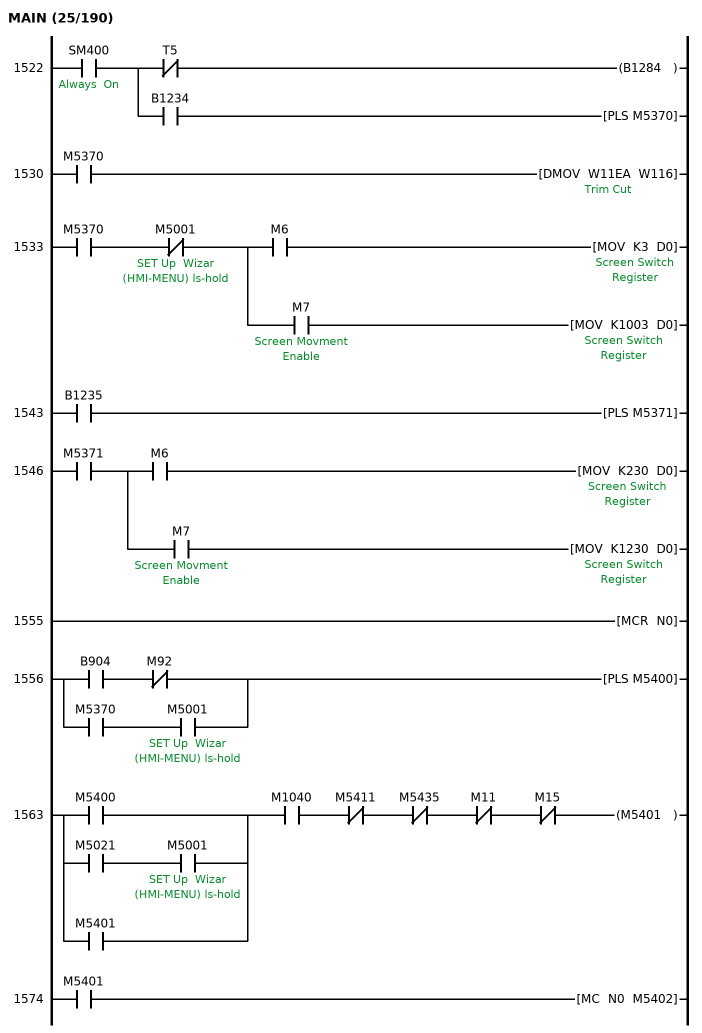
[picture p24: ladder of MAIN, rungs at steps 1522 to 1574]
1522  LD      SM400  ; Always  On
      MPS
      ANI     T5
      OUT     B1284
      MPP
      AND     B1234
      PLS     M5370
1530  LD      M5370
      DMOV    W11EA W116
1533  LD      M5370
      ANI     M5001  ; SET Up  Wizar (HMI-MENU) ls-hold
      MPS
      AND     M6
      MOV     K3 D0
      MPP
      AND     M7  ; Screen Movment Enable
      MOV     K1003 D0
1543  LD      B1235
      PLS     M5371
1546  LD      M5371
      MPS
      AND     M6
      MOV     K230 D0
      MPP
      AND     M7  ; Screen Movment Enable
      MOV     K1230 D0
1555  MCR     N0
1556  LD      B904
      ANI     M92
      LD      M5370
      AND     M5001  ; SET Up  Wizar (HMI-MENU) ls-hold
      ORB
      PLS     M5400
1563  LD      M5400
      LD      M5021
      AND     M5001  ; SET Up  Wizar (HMI-MENU) ls-hold
      ORB
      OR      M5401
      AND     M1040
      ANI     M5411
      ANI     M5435
      ANI     M11
      ANI     M15
      OUT     M5401
1574  LD      M5401
      MC      N0 M5402
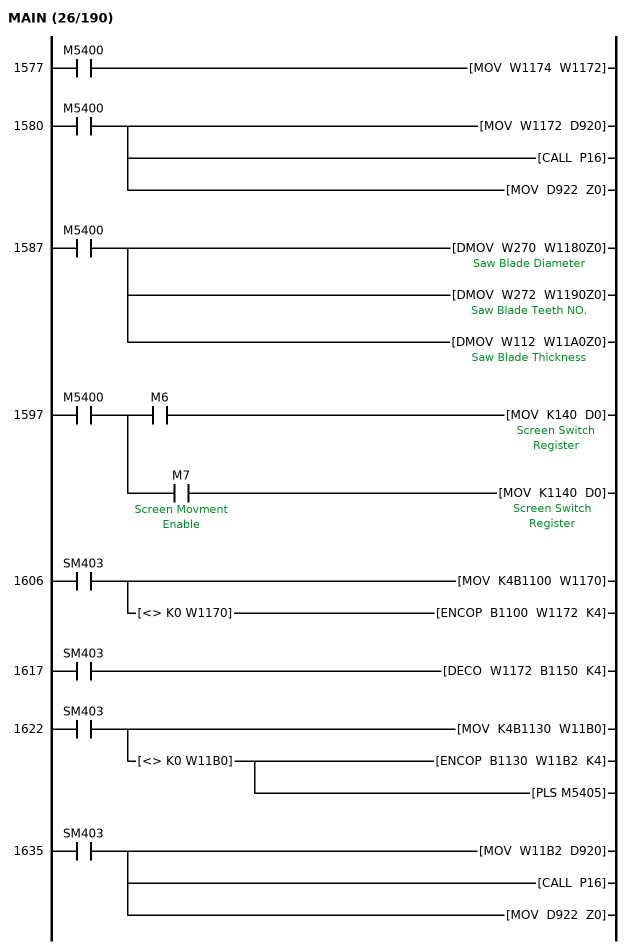
1577  LD      M5400
      MOV     W1174 W1172
1580  LD      M5400
      MOV     W1172 D920
      CALL    P16
      MOV     D922 Z0
1587  LD      M5400
      DMOV    W270 W1180Z0  ; Saw Blade Diameter
      DMOV    W272 W1190Z0  ; Saw Blade Teeth NO.
      DMOV    W112 W11A0Z0  ; Saw Blade Thickness
1597  LD      M5400
      MPS
      AND     M6
      MOV     K140 D0
      MPP
      AND     M7  ; Screen Movment Enable
      MOV     K1140 D0
1606  LD      SM403
      MOV     K4B1100 W1170
      AND<>   K0 W1170
      ENCOP   B1100 W1172 K4
1617  LD      SM403
      DECO    W1172 B1150 K4
1622  LD      SM403
      MOV     K4B1130 W11B0
      AND<>   K0 W11B0
      ENCOP   B1130 W11B2 K4
      PLS     M5405
1635  LD      SM403
      MOV     W11B2 D920
      CALL    P16
      MOV     D922 Z0
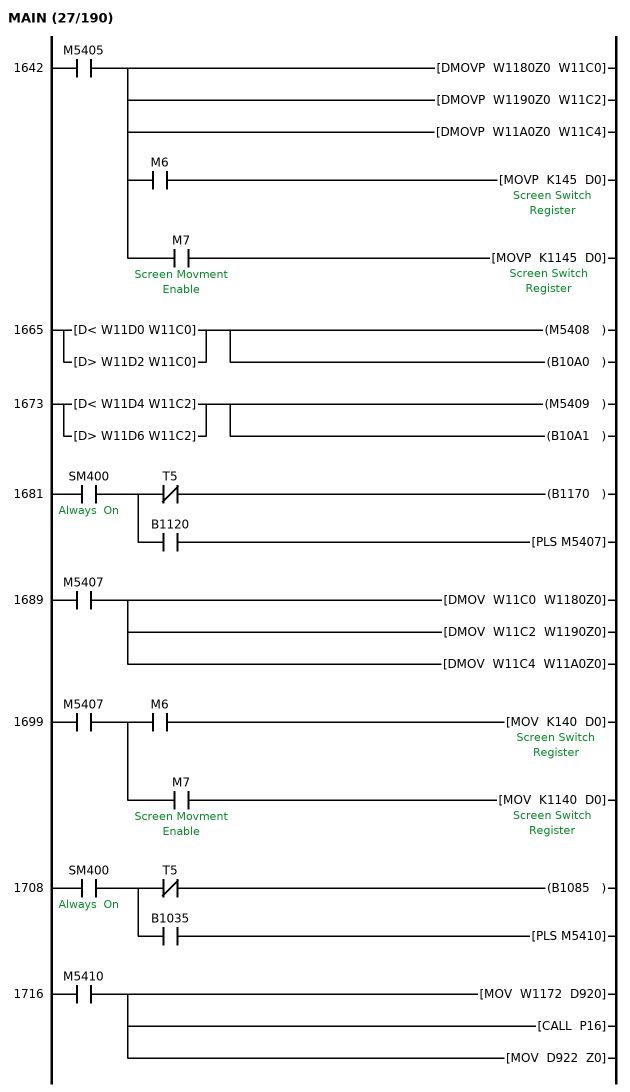
1642  LD      M5405
      DMOVP   W1180Z0 W11C0
      DMOVP   W1190Z0 W11C2
      DMOVP   W11A0Z0 W11C4
      MPS
      AND     M6
      MOVP    K145 D0
      MPP
      AND     M7  ; Screen Movment Enable
      MOVP    K1145 D0
1665  LDD<    W11D0 W11C0
      ORD>    W11D2 W11C0
      OUT     M5408
      OUT     B10A0
1673  LDD<    W11D4 W11C2
      ORD>    W11D6 W11C2
      OUT     M5409
      OUT     B10A1
1681  LD      SM400  ; Always  On
      MPS
      ANI     T5
      OUT     B1170
      MPP
      AND     B1120
      PLS     M5407
1689  LD      M5407
      DMOV    W11C0 W1180Z0
      DMOV    W11C2 W1190Z0
      DMOV    W11C4 W11A0Z0
1699  LD      M5407
      MPS
      AND     M6
      MOV     K140 D0
      MPP
      AND     M7  ; Screen Movment Enable
      MOV     K1140 D0
1708  LD      SM400  ; Always  On
      MPS
      ANI     T5
      OUT     B1085
      MPP
      AND     B1035
      PLS     M5410
1716  LD      M5410
      MOV     W1172 D920
      CALL    P16
      MOV     D922 Z0
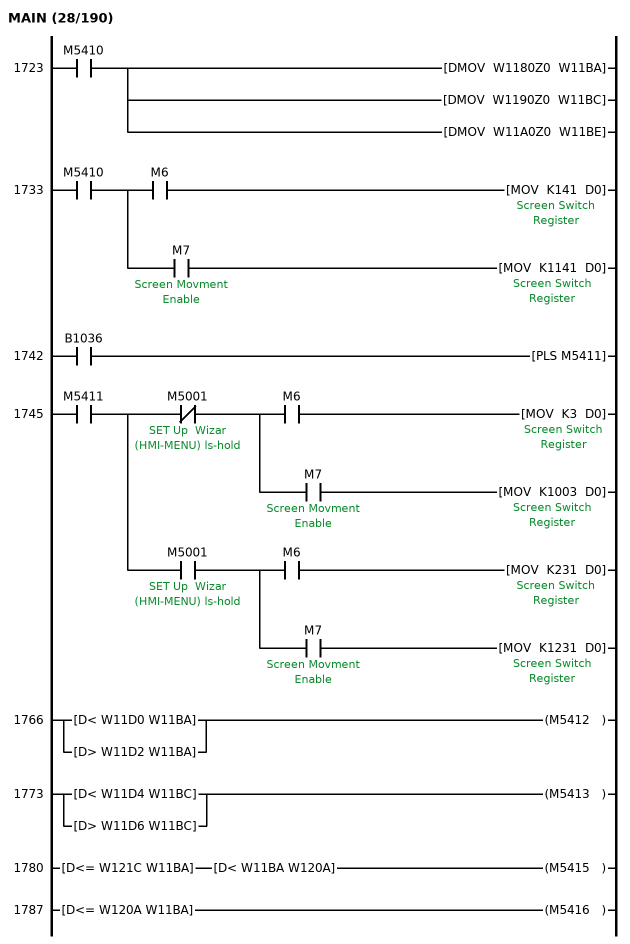
1723  LD      M5410
      DMOV    W1180Z0 W11BA
      DMOV    W1190Z0 W11BC
      DMOV    W11A0Z0 W11BE
1733  LD      M5410
      MPS
      AND     M6
      MOV     K141 D0
      MPP
      AND     M7  ; Screen Movment Enable
      MOV     K1141 D0
1742  LD      B1036
      PLS     M5411
1745  LD      M5411
      MPS
      ANI     M5001  ; SET Up  Wizar (HMI-MENU) ls-hold
      MPS
      AND     M6
      MOV     K3 D0
      MPP
      AND     M7  ; Screen Movment Enable
      MOV     K1003 D0
      MPP
      AND     M5001  ; SET Up  Wizar (HMI-MENU) ls-hold
      MPS
      AND     M6
      MOV     K231 D0
      MPP
      AND     M7  ; Screen Movment Enable
      MOV     K1231 D0
1766  LDD<    W11D0 W11BA
      ORD>    W11D2 W11BA
      OUT     M5412
1773  LDD<    W11D4 W11BC
      ORD>    W11D6 W11BC
      OUT     M5413
1780  LDD<=   W121C W11BA
      ANDD<   W11BA W120A
      OUT     M5415
1787  LDD<=   W120A W11BA
      OUT     M5416
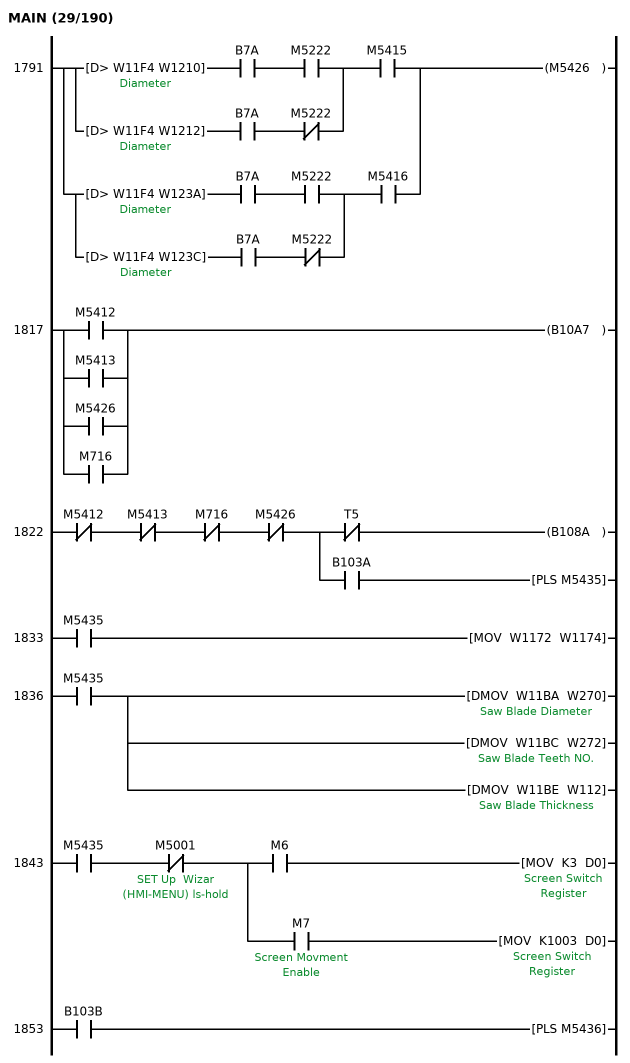
1791  LDD>    W11F4 W1210  ; Diameter
      AND     B7A
      AND     M5222
      LDD>    W11F4 W1212  ; Diameter
      AND     B7A
      ANI     M5222
      ORB
      AND     M5415
      LDD>    W11F4 W123A  ; Diameter
      AND     B7A
      AND     M5222
      LDD>    W11F4 W123C  ; Diameter
      AND     B7A
      ANI     M5222
      ORB
      AND     M5416
      ORB
      OUT     M5426
1817  LD      M5412
      OR      M5413
      OR      M5426
      OR      M716
      OUT     B10A7
1822  LDI     M5412
      ANI     M5413
      ANI     M716
      ANI     M5426
      MPS
      ANI     T5
      OUT     B108A
      MPP
      AND     B103A
      PLS     M5435
1833  LD      M5435
      MOV     W1172 W1174
1836  LD      M5435
      DMOV    W11BA W270
      DMOV    W11BC W272
      DMOV    W11BE W112
1843  LD      M5435
      ANI     M5001  ; SET Up  Wizar (HMI-MENU) ls-hold
      MPS
      AND     M6
      MOV     K3 D0
      MPP
      AND     M7  ; Screen Movment Enable
      MOV     K1003 D0
1853  LD      B103B
      PLS     M5436
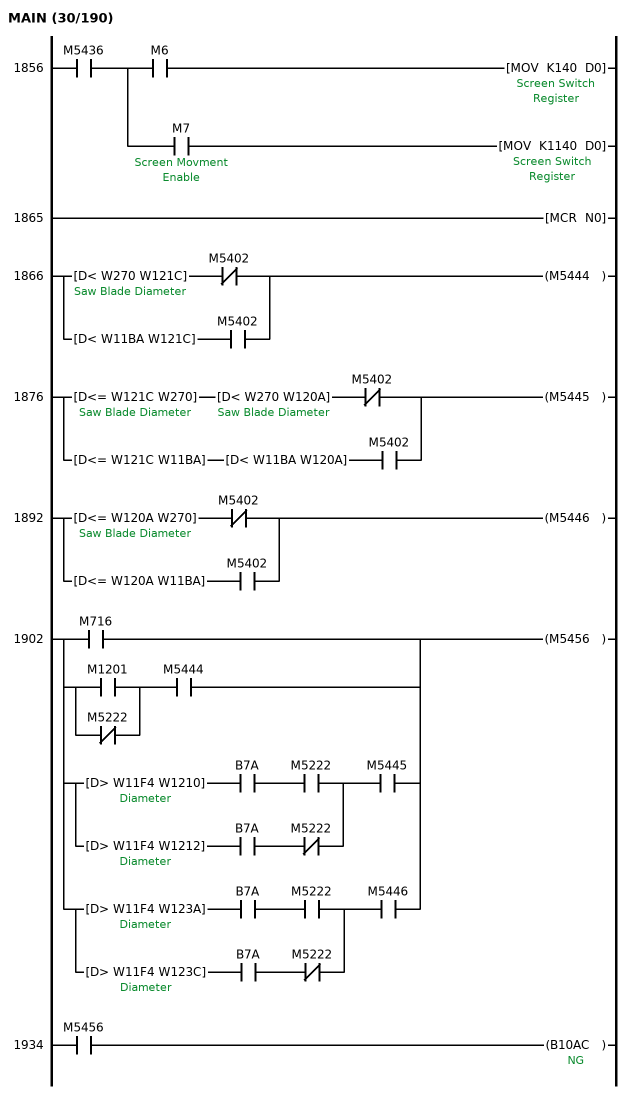
1856  LD      M5436
      MPS
      AND     M6
      MOV     K140 D0
      MPP
      AND     M7  ; Screen Movment Enable
      MOV     K1140 D0
1865  MCR     N0
1866  LDD<    W270 W121C  ; Saw Blade Diameter
      ANI     M5402
      LDD<    W11BA W121C
      AND     M5402
      ORB
      OUT     M5444
1876  LDD<=   W121C W270  ; Saw Blade Diameter
      ANDD<   W270 W120A  ; Saw Blade Diameter
      ANI     M5402
      LDD<=   W121C W11BA
      ANDD<   W11BA W120A
      AND     M5402
      ORB
      OUT     M5445
1892  LDD<=   W120A W270  ; Saw Blade Diameter
      ANI     M5402
      LDD<=   W120A W11BA
      AND     M5402
      ORB
      OUT     M5446
1902  LD      M716
      LD      M1201
      ORI     M5222
      AND     M5444
      ORB
      LDD>    W11F4 W1210  ; Diameter
      AND     B7A
      AND     M5222
      LDD>    W11F4 W1212  ; Diameter
      AND     B7A
      ANI     M5222
      ORB
      AND     M5445
      ORB
      LDD>    W11F4 W123A  ; Diameter
      AND     B7A
      AND     M5222
      LDD>    W11F4 W123C  ; Diameter
      AND     B7A
      ANI     M5222
      ORB
      AND     M5446
      ORB
      OUT     M5456
1934  LD      M5456
      OUT     B10AC  ; NG
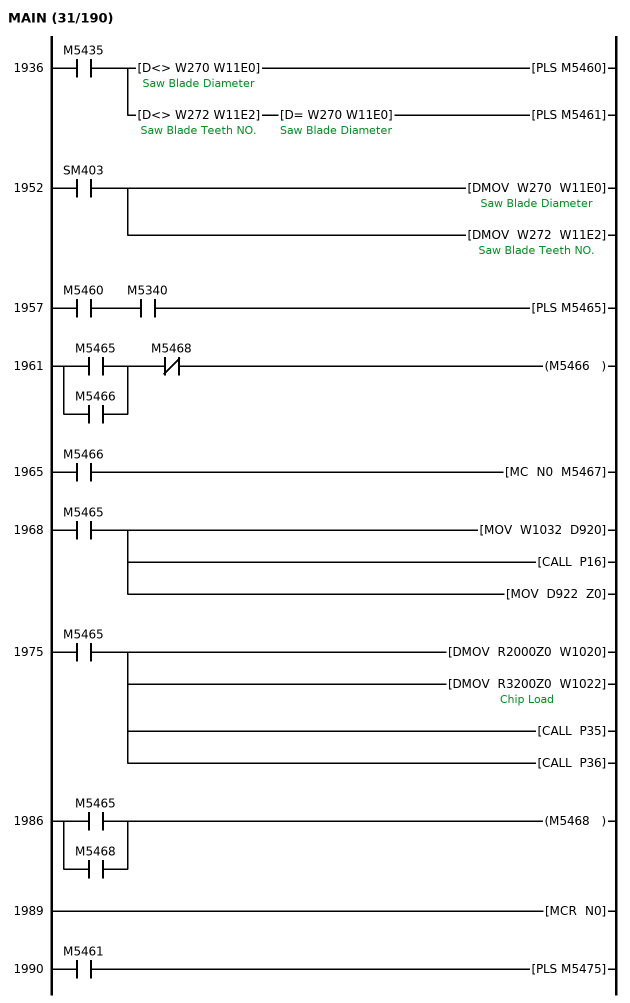
1936  LD      M5435
      MPS
      ANDD<>  W270 W11E0  ; Saw Blade Diameter
      PLS     M5460
      MPP
      ANDD<>  W272 W11E2  ; Saw Blade Teeth NO.
      ANDD=   W270 W11E0  ; Saw Blade Diameter
      PLS     M5461
1952  LD      SM403
      DMOV    W270 W11E0
      DMOV    W272 W11E2
1957  LD      M5460
      AND     M5340
      PLS     M5465
1961  LD      M5465
      OR      M5466
      ANI     M5468
      OUT     M5466
1965  LD      M5466
      MC      N0 M5467
1968  LD      M5465
      MOV     W1032 D920
      CALL    P16
      MOV     D922 Z0
1975  LD      M5465
      DMOV    R2000Z0 W1020
      DMOV    R3200Z0 W1022
      CALL    P35
      CALL    P36
1986  LD      M5465
      OR      M5468
      OUT     M5468
1989  MCR     N0
1990  LD      M5461
      PLS     M5475
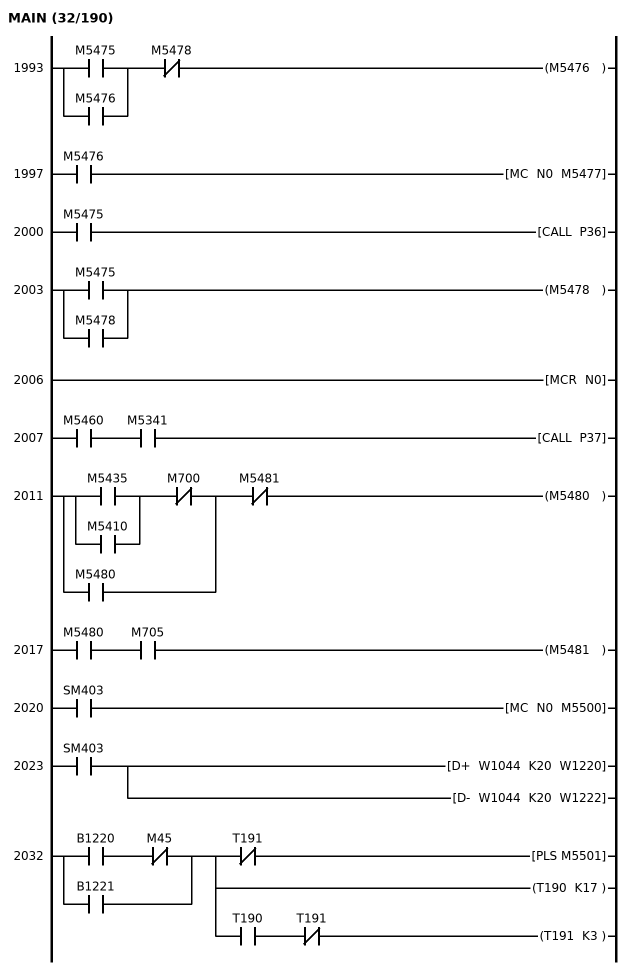
1993  LD      M5475
      OR      M5476
      ANI     M5478
      OUT     M5476
1997  LD      M5476
      MC      N0 M5477
2000  LD      M5475
      CALL    P36
2003  LD      M5475
      OR      M5478
      OUT     M5478
2006  MCR     N0
2007  LD      M5460
      AND     M5341
      CALL    P37
2011  LD      M5435
      OR      M5410
      ANI     M700
      OR      M5480
      ANI     M5481
      OUT     M5480
2017  LD      M5480
      AND     M705
      OUT     M5481
2020  LD      SM403
      MC      N0 M5500
2023  LD      SM403
      D+      W1044 K20 W1220
      D-      W1044 K20 W1222
2032  LD      B1220
      ANI     M45
      OR      B1221
      MPS
      ANI     T191
      PLS     M5501
      MPP
      OUT     T190 K17
      AND     T190
      ANI     T191
      OUT     T191 K3
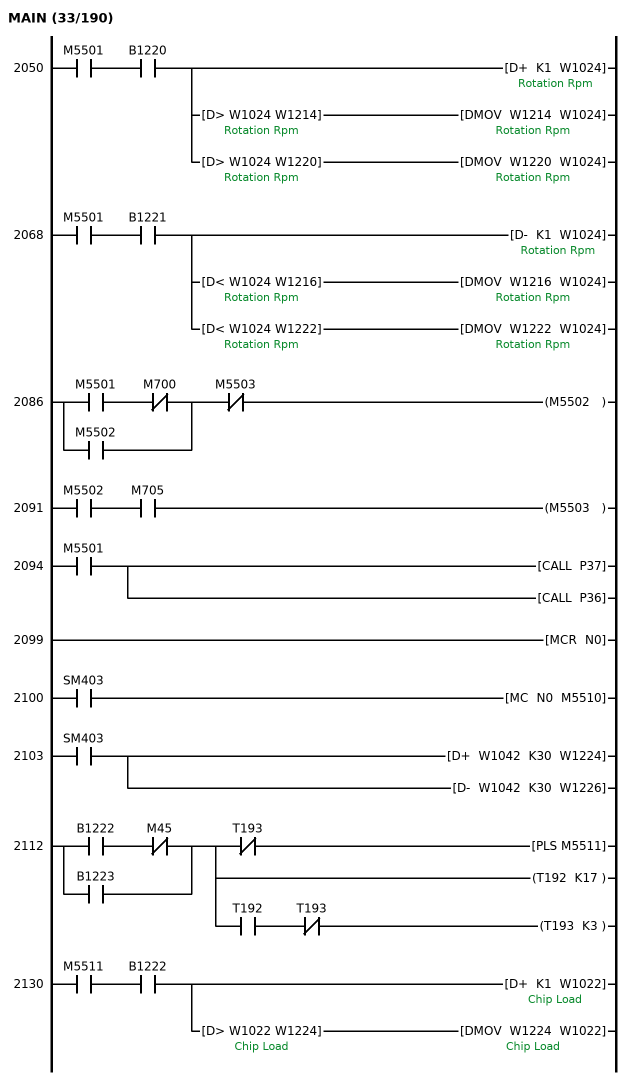
2050  LD      M5501
      AND     B1220
      D+      K1 W1024
      MPS
      ANDD>   W1024 W1214  ; Rotation Rpm
      DMOV    W1214 W1024
      MPP
      ANDD>   W1024 W1220  ; Rotation Rpm
      DMOV    W1220 W1024
2068  LD      M5501
      AND     B1221
      D-      K1 W1024
      MPS
      ANDD<   W1024 W1216  ; Rotation Rpm
      DMOV    W1216 W1024
      MPP
      ANDD<   W1024 W1222  ; Rotation Rpm
      DMOV    W1222 W1024
2086  LD      M5501
      ANI     M700
      OR      M5502
      ANI     M5503
      OUT     M5502
2091  LD      M5502
      AND     M705
      OUT     M5503
2094  LD      M5501
      CALL    P37
      CALL    P36
2099  MCR     N0
2100  LD      SM403
      MC      N0 M5510
2103  LD      SM403
      D+      W1042 K30 W1224
      D-      W1042 K30 W1226
2112  LD      B1222
      ANI     M45
      OR      B1223
      MPS
      ANI     T193
      PLS     M5511
      MPP
      OUT     T192 K17
      AND     T192
      ANI     T193
      OUT     T193 K3
2130  LD      M5511
      AND     B1222
      D+      K1 W1022
      ANDD>   W1022 W1224  ; Chip Load
      DMOV    W1224 W1022
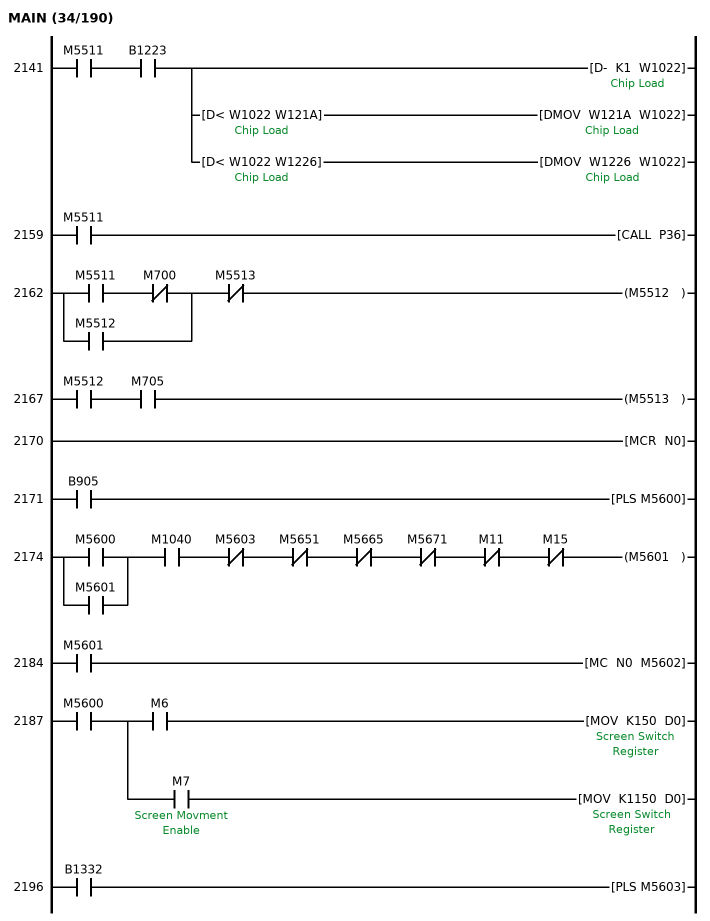
2141  LD      M5511
      AND     B1223
      D-      K1 W1022
      MPS
      ANDD<   W1022 W121A  ; Chip Load
      DMOV    W121A W1022
      MPP
      ANDD<   W1022 W1226  ; Chip Load
      DMOV    W1226 W1022
2159  LD      M5511
      CALL    P36
2162  LD      M5511
      ANI     M700
      OR      M5512
      ANI     M5513
      OUT     M5512
2167  LD      M5512
      AND     M705
      OUT     M5513
2170  MCR     N0
2171  LD      B905
      PLS     M5600
2174  LD      M5600
      OR      M5601
      AND     M1040
      ANI     M5603
      ANI     M5651
      ANI     M5665
      ANI     M5671
      ANI     M11
      ANI     M15
      OUT     M5601
2184  LD      M5601
      MC      N0 M5602
2187  LD      M5600
      MPS
      AND     M6
      MOV     K150 D0
      MPP
      AND     M7  ; Screen Movment Enable
      MOV     K1150 D0
2196  LD      B1332
      PLS     M5603
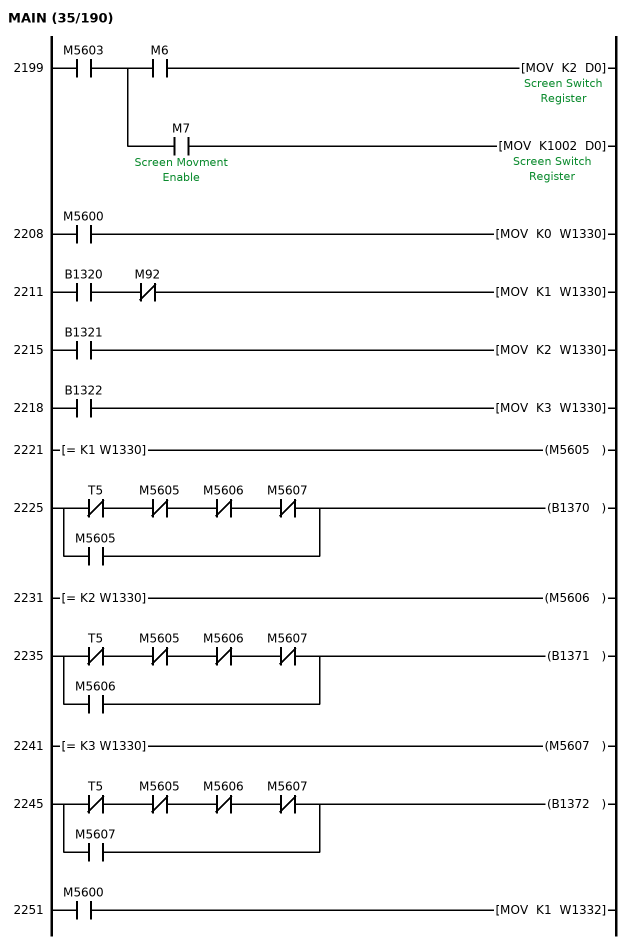
2199  LD      M5603
      MPS
      AND     M6
      MOV     K2 D0
      MPP
      AND     M7  ; Screen Movment Enable
      MOV     K1002 D0
2208  LD      M5600
      MOV     K0 W1330
2211  LD      B1320
      ANI     M92
      MOV     K1 W1330
2215  LD      B1321
      MOV     K2 W1330
2218  LD      B1322
      MOV     K3 W1330
2221  LD=     K1 W1330
      OUT     M5605
2225  LDI     T5
      ANI     M5605
      ANI     M5606
      ANI     M5607
      OR      M5605
      OUT     B1370
2231  LD=     K2 W1330
      OUT     M5606
2235  LDI     T5
      ANI     M5605
      ANI     M5606
      ANI     M5607
      OR      M5606
      OUT     B1371
2241  LD=     K3 W1330
      OUT     M5607
2245  LDI     T5
      ANI     M5605
      ANI     M5606
      ANI     M5607
      OR      M5607
      OUT     B1372
2251  LD      M5600
      MOV     K1 W1332
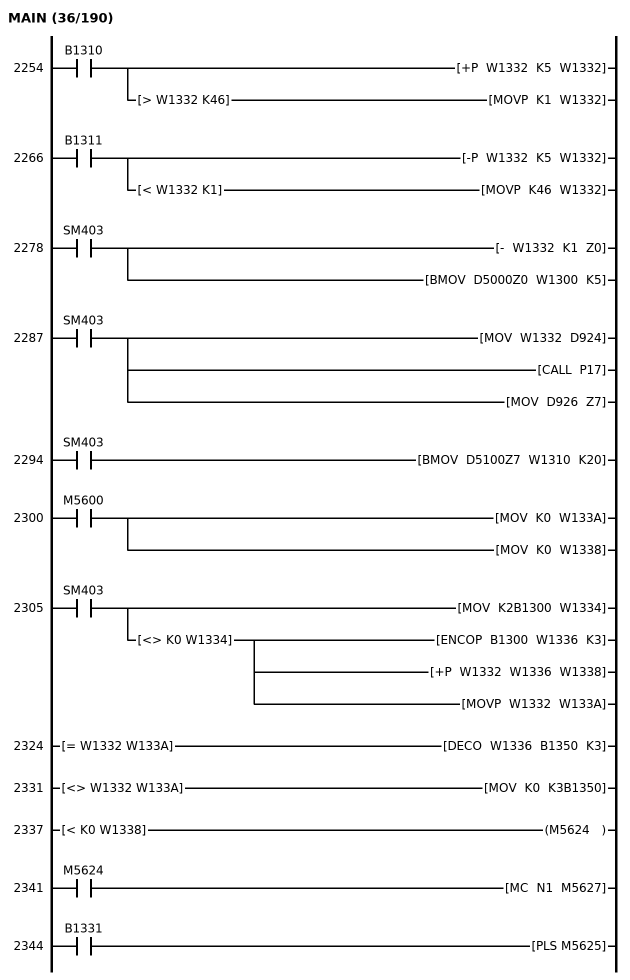
2254  LD      B1310
      +P      W1332 K5 W1332
      AND>    W1332 K46
      MOVP    K1 W1332
2266  LD      B1311
      -P      W1332 K5 W1332
      AND<    W1332 K1
      MOVP    K46 W1332
2278  LD      SM403
      -       W1332 K1 Z0
      BMOV    D5000Z0 W1300 K5
2287  LD      SM403
      MOV     W1332 D924
      CALL    P17
      MOV     D926 Z7
2294  LD      SM403
      BMOV    D5100Z7 W1310 K20
2300  LD      M5600
      MOV     K0 W133A
      MOV     K0 W1338
2305  LD      SM403
      MOV     K2B1300 W1334
      AND<>   K0 W1334
      ENCOP   B1300 W1336 K3
      +P      W1332 W1336 W1338
      MOVP    W1332 W133A
2324  LD=     W1332 W133A
      DECO    W1336 B1350 K3
2331  LD<>    W1332 W133A
      MOV     K0 K3B1350
2337  LD<     K0 W1338
      OUT     M5624
2341  LD      M5624
      MC      N1 M5627
2344  LD      B1331
      PLS     M5625
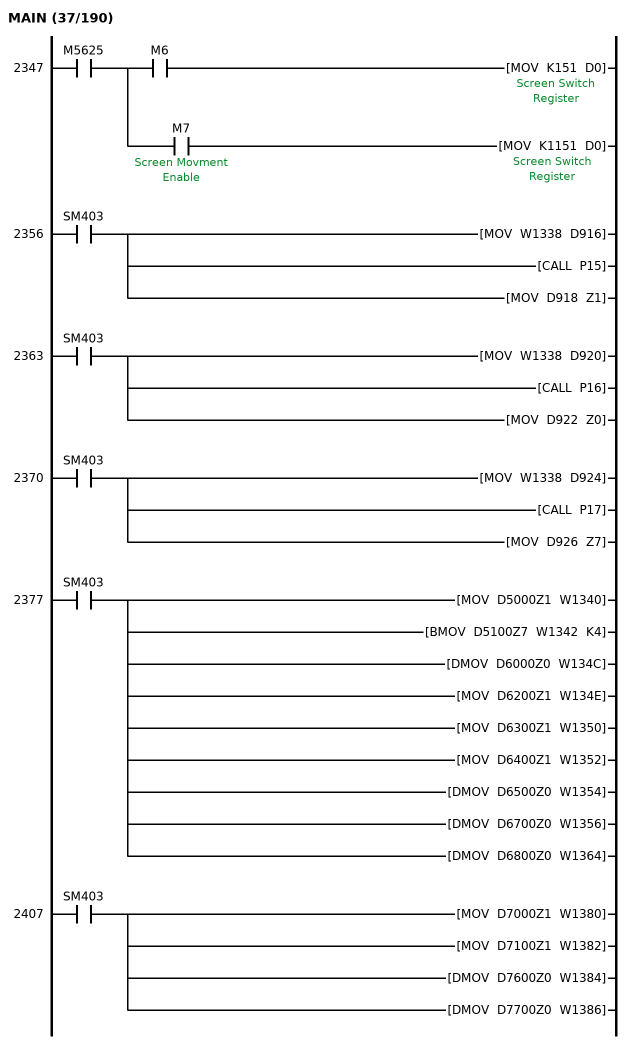
2347  LD      M5625
      MPS
      AND     M6
      MOV     K151 D0
      MPP
      AND     M7  ; Screen Movment Enable
      MOV     K1151 D0
2356  LD      SM403
      MOV     W1338 D916
      CALL    P15
      MOV     D918 Z1
2363  LD      SM403
      MOV     W1338 D920
      CALL    P16
      MOV     D922 Z0
2370  LD      SM403
      MOV     W1338 D924
      CALL    P17
      MOV     D926 Z7
2377  LD      SM403
      MOV     D5000Z1 W1340
      BMOV    D5100Z7 W1342 K4
      DMOV    D6000Z0 W134C
      MOV     D6200Z1 W134E
      MOV     D6300Z1 W1350
      MOV     D6400Z1 W1352
      DMOV    D6500Z0 W1354
      DMOV    D6700Z0 W1356
      DMOV    D6800Z0 W1364
2407  LD      SM403
      MOV     D7000Z1 W1380
      MOV     D7100Z1 W1382
      DMOV    D7600Z0 W1384
      DMOV    D7700Z0 W1386
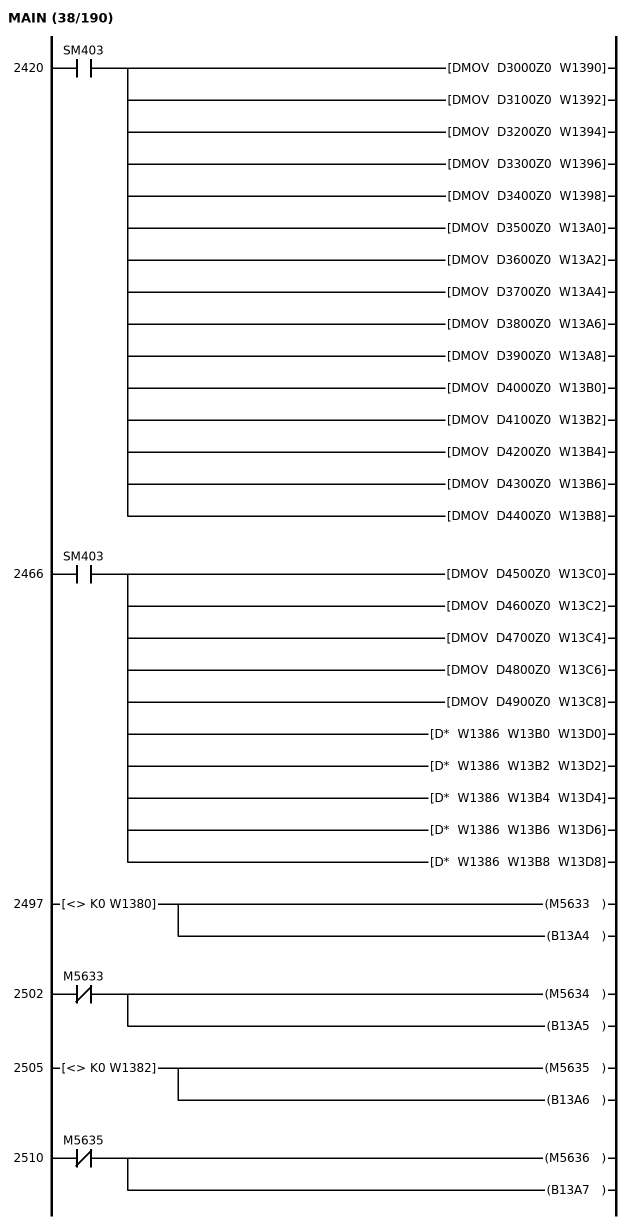
2420  LD      SM403
      DMOV    D3000Z0 W1390
      DMOV    D3100Z0 W1392
      DMOV    D3200Z0 W1394
      DMOV    D3300Z0 W1396
      DMOV    D3400Z0 W1398
      DMOV    D3500Z0 W13A0
      DMOV    D3600Z0 W13A2
      DMOV    D3700Z0 W13A4
      DMOV    D3800Z0 W13A6
      DMOV    D3900Z0 W13A8
      DMOV    D4000Z0 W13B0
      DMOV    D4100Z0 W13B2
      DMOV    D4200Z0 W13B4
      DMOV    D4300Z0 W13B6
      DMOV    D4400Z0 W13B8
2466  LD      SM403
      DMOV    D4500Z0 W13C0
      DMOV    D4600Z0 W13C2
      DMOV    D4700Z0 W13C4
      DMOV    D4800Z0 W13C6
      DMOV    D4900Z0 W13C8
      D*      W1386 W13B0 W13D0
      D*      W1386 W13B2 W13D2
      D*      W1386 W13B4 W13D4
      D*      W1386 W13B6 W13D6
      D*      W1386 W13B8 W13D8
2497  LD<>    K0 W1380
      OUT     M5633
      OUT     B13A4
2502  LDI     M5633
      OUT     M5634
      OUT     B13A5
2505  LD<>    K0 W1382
      OUT     M5635
      OUT     B13A6
2510  LDI     M5635
      OUT     M5636
      OUT     B13A7
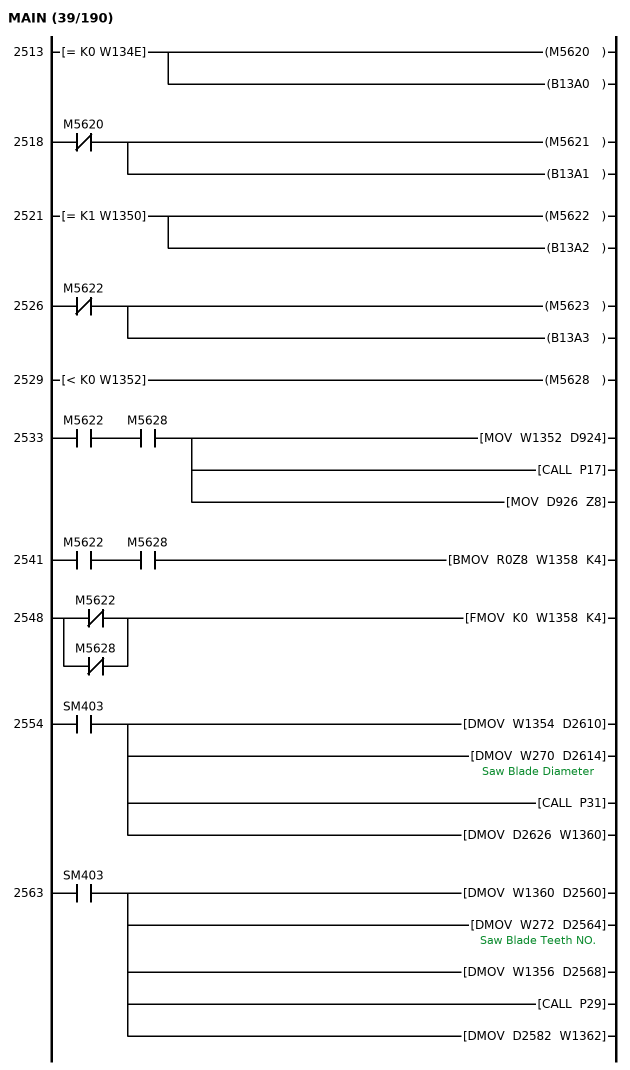
2513  LD=     K0 W134E
      OUT     M5620
      OUT     B13A0
2518  LDI     M5620
      OUT     M5621
      OUT     B13A1
2521  LD=     K1 W1350
      OUT     M5622
      OUT     B13A2
2526  LDI     M5622
      OUT     M5623
      OUT     B13A3
2529  LD<     K0 W1352
      OUT     M5628
2533  LD      M5622
      AND     M5628
      MOV     W1352 D924
      CALL    P17
      MOV     D926 Z8
2541  LD      M5622
      AND     M5628
      BMOV    R0Z8 W1358 K4
2548  LDI     M5622
      ORI     M5628
      FMOV    K0 W1358 K4
2554  LD      SM403
      DMOV    W1354 D2610
      DMOV    W270 D2614
      CALL    P31
      DMOV    D2626 W1360
2563  LD      SM403
      DMOV    W1360 D2560
      DMOV    W272 D2564
      DMOV    W1356 D2568
      CALL    P29
      DMOV    D2582 W1362
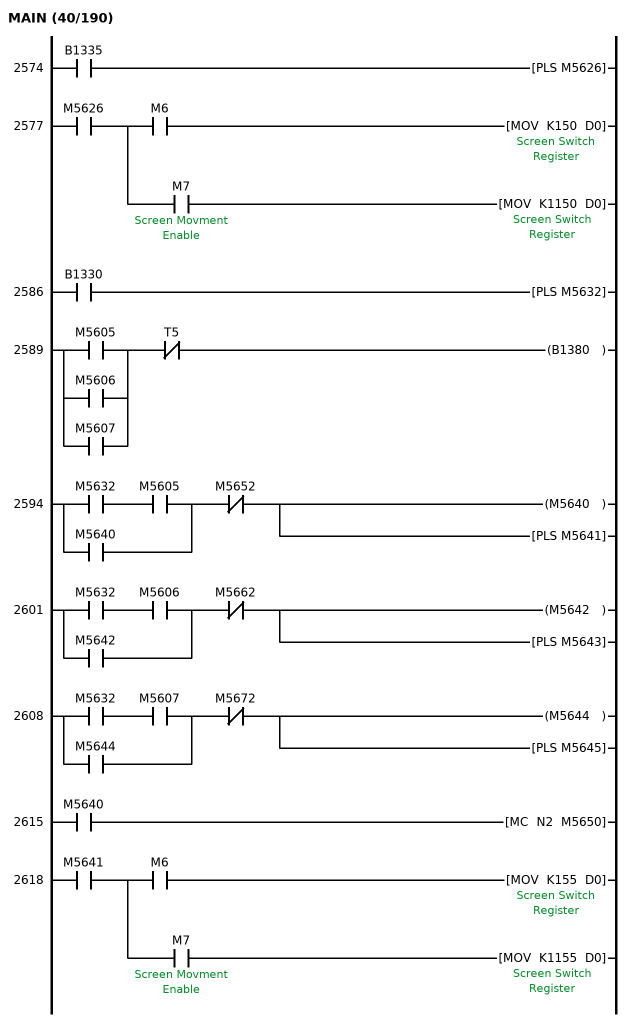
2574  LD      B1335
      PLS     M5626
2577  LD      M5626
      MPS
      AND     M6
      MOV     K150 D0
      MPP
      AND     M7  ; Screen Movment Enable
      MOV     K1150 D0
2586  LD      B1330
      PLS     M5632
2589  LD      M5605
      OR      M5606
      OR      M5607
      ANI     T5
      OUT     B1380
2594  LD      M5632
      AND     M5605
      OR      M5640
      ANI     M5652
      OUT     M5640
      PLS     M5641
2601  LD      M5632
      AND     M5606
      OR      M5642
      ANI     M5662
      OUT     M5642
      PLS     M5643
2608  LD      M5632
      AND     M5607
      OR      M5644
      ANI     M5672
      OUT     M5644
      PLS     M5645
2615  LD      M5640
      MC      N2 M5650
2618  LD      M5641
      MPS
      AND     M6
      MOV     K155 D0
      MPP
      AND     M7  ; Screen Movment Enable
      MOV     K1155 D0
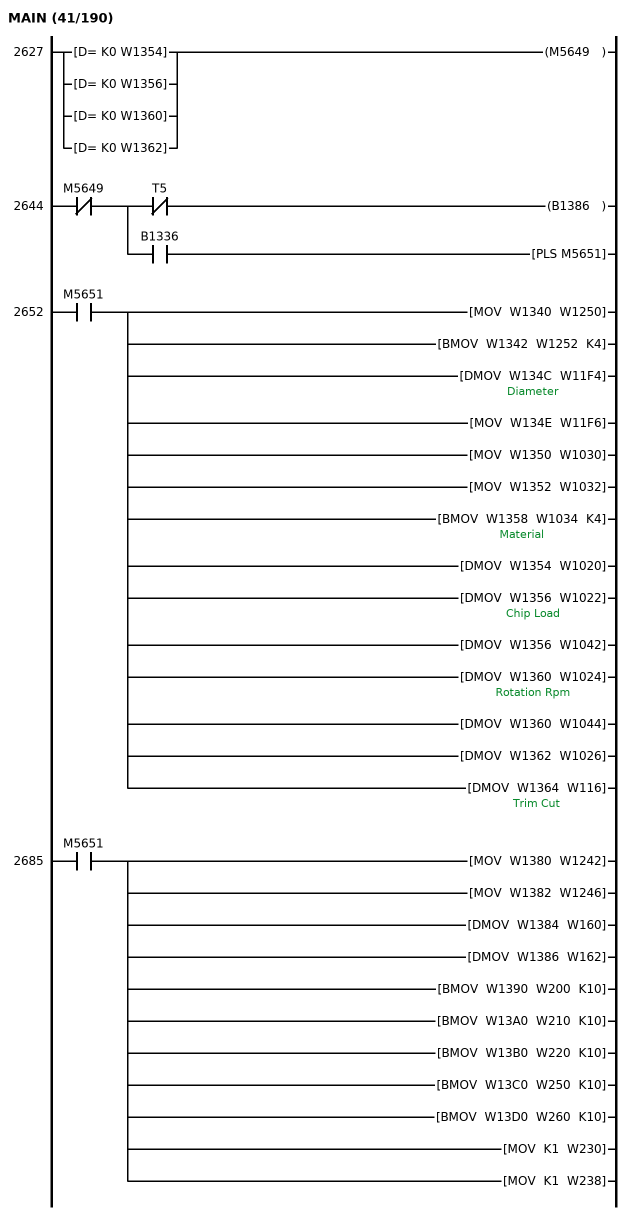
2627  LDD=    K0 W1354
      ORD=    K0 W1356
      ORD=    K0 W1360
      ORD=    K0 W1362
      OUT     M5649
2644  LDI     M5649
      MPS
      ANI     T5
      OUT     B1386
      MPP
      AND     B1336
      PLS     M5651
2652  LD      M5651
      MOV     W1340 W1250
      BMOV    W1342 W1252 K4
      DMOV    W134C W11F4
      MOV     W134E W11F6
      MOV     W1350 W1030
      MOV     W1352 W1032
      BMOV    W1358 W1034 K4
      DMOV    W1354 W1020
      DMOV    W1356 W1022
      DMOV    W1356 W1042
      DMOV    W1360 W1024
      DMOV    W1360 W1044
      DMOV    W1362 W1026
      DMOV    W1364 W116
2685  LD      M5651
      MOV     W1380 W1242
      MOV     W1382 W1246
      DMOV    W1384 W160
      DMOV    W1386 W162
      BMOV    W1390 W200 K10
      BMOV    W13A0 W210 K10
      BMOV    W13B0 W220 K10
      BMOV    W13C0 W250 K10
      BMOV    W13D0 W260 K10
      MOV     K1 W230
      MOV     K1 W238
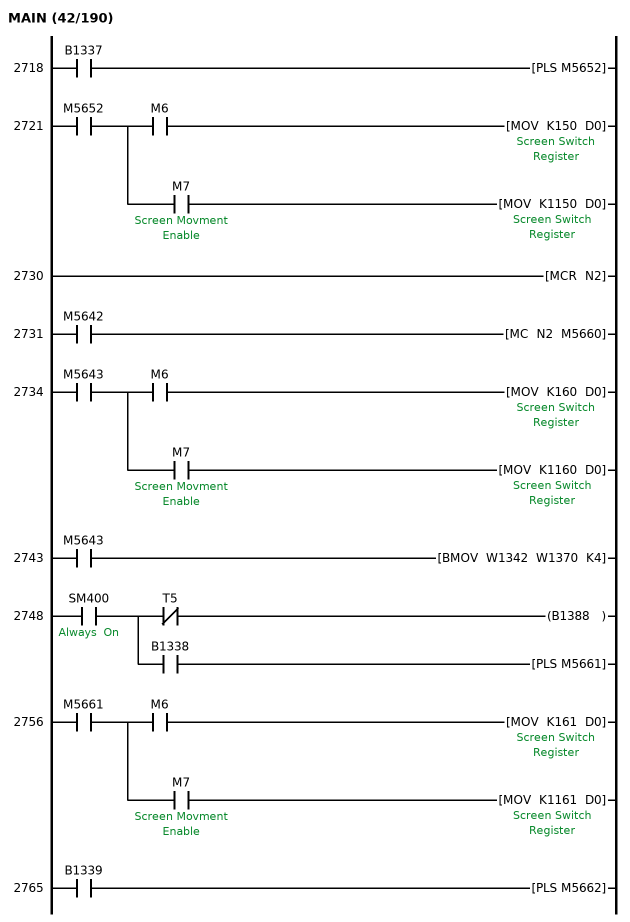
2718  LD      B1337
      PLS     M5652
2721  LD      M5652
      MPS
      AND     M6
      MOV     K150 D0
      MPP
      AND     M7  ; Screen Movment Enable
      MOV     K1150 D0
2730  MCR     N2
2731  LD      M5642
      MC      N2 M5660
2734  LD      M5643
      MPS
      AND     M6
      MOV     K160 D0
      MPP
      AND     M7  ; Screen Movment Enable
      MOV     K1160 D0
2743  LD      M5643
      BMOV    W1342 W1370 K4
2748  LD      SM400  ; Always  On
      MPS
      ANI     T5
      OUT     B1388
      MPP
      AND     B1338
      PLS     M5661
2756  LD      M5661
      MPS
      AND     M6
      MOV     K161 D0
      MPP
      AND     M7  ; Screen Movment Enable
      MOV     K1161 D0
2765  LD      B1339
      PLS     M5662
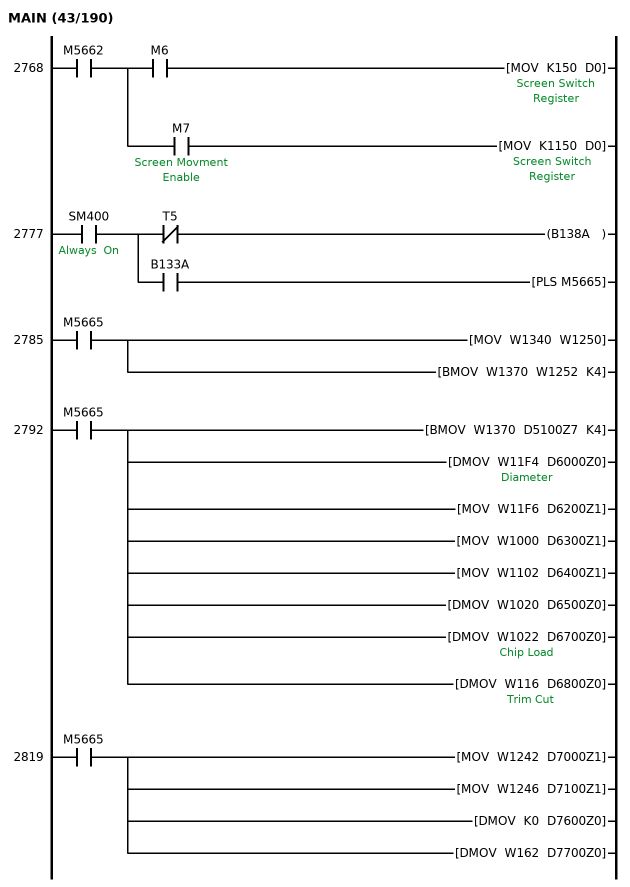
2768  LD      M5662
      MPS
      AND     M6
      MOV     K150 D0
      MPP
      AND     M7  ; Screen Movment Enable
      MOV     K1150 D0
2777  LD      SM400  ; Always  On
      MPS
      ANI     T5
      OUT     B138A
      MPP
      AND     B133A
      PLS     M5665
2785  LD      M5665
      MOV     W1340 W1250
      BMOV    W1370 W1252 K4
2792  LD      M5665
      BMOV    W1370 D5100Z7 K4
      DMOV    W11F4 D6000Z0
      MOV     W11F6 D6200Z1
      MOV     W1000 D6300Z1
      MOV     W1102 D6400Z1
      DMOV    W1020 D6500Z0
      DMOV    W1022 D6700Z0
      DMOV    W116 D6800Z0
2819  LD      M5665
      MOV     W1242 D7000Z1
      MOV     W1246 D7100Z1
      DMOV    K0 D7600Z0
      DMOV    W162 D7700Z0
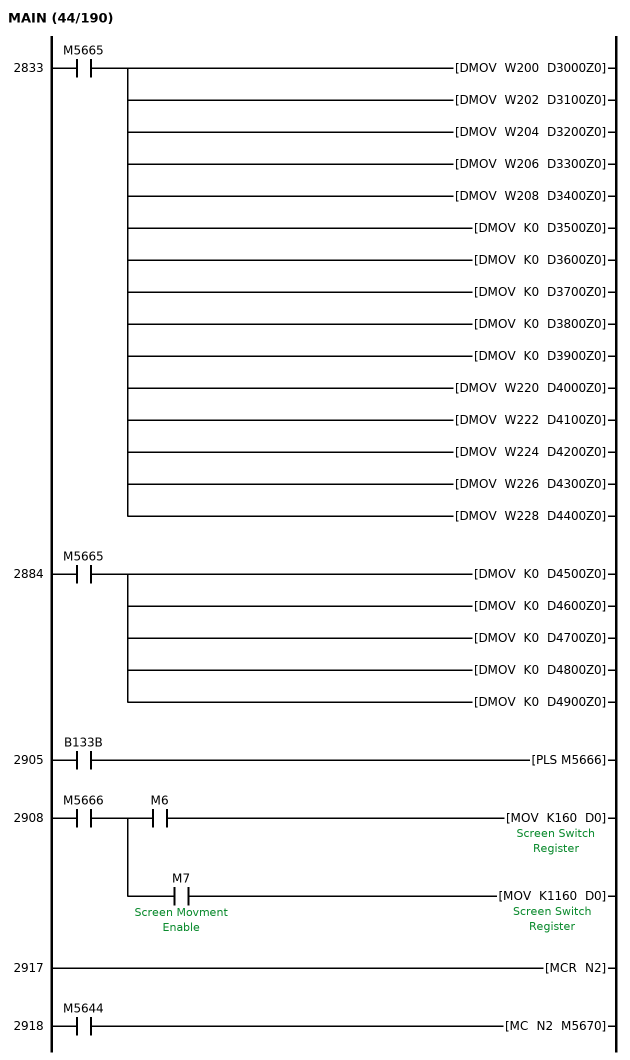
2833  LD      M5665
      DMOV    W200 D3000Z0
      DMOV    W202 D3100Z0
      DMOV    W204 D3200Z0
      DMOV    W206 D3300Z0
      DMOV    W208 D3400Z0
      DMOV    K0 D3500Z0
      DMOV    K0 D3600Z0
      DMOV    K0 D3700Z0
      DMOV    K0 D3800Z0
      DMOV    K0 D3900Z0
      DMOV    W220 D4000Z0
      DMOV    W222 D4100Z0
      DMOV    W224 D4200Z0
      DMOV    W226 D4300Z0
      DMOV    W228 D4400Z0
2884  LD      M5665
      DMOV    K0 D4500Z0
      DMOV    K0 D4600Z0
      DMOV    K0 D4700Z0
      DMOV    K0 D4800Z0
      DMOV    K0 D4900Z0
2905  LD      B133B
      PLS     M5666
2908  LD      M5666
      MPS
      AND     M6
      MOV     K160 D0
      MPP
      AND     M7  ; Screen Movment Enable
      MOV     K1160 D0
2917  MCR     N2
2918  LD      M5644
      MC      N2 M5670
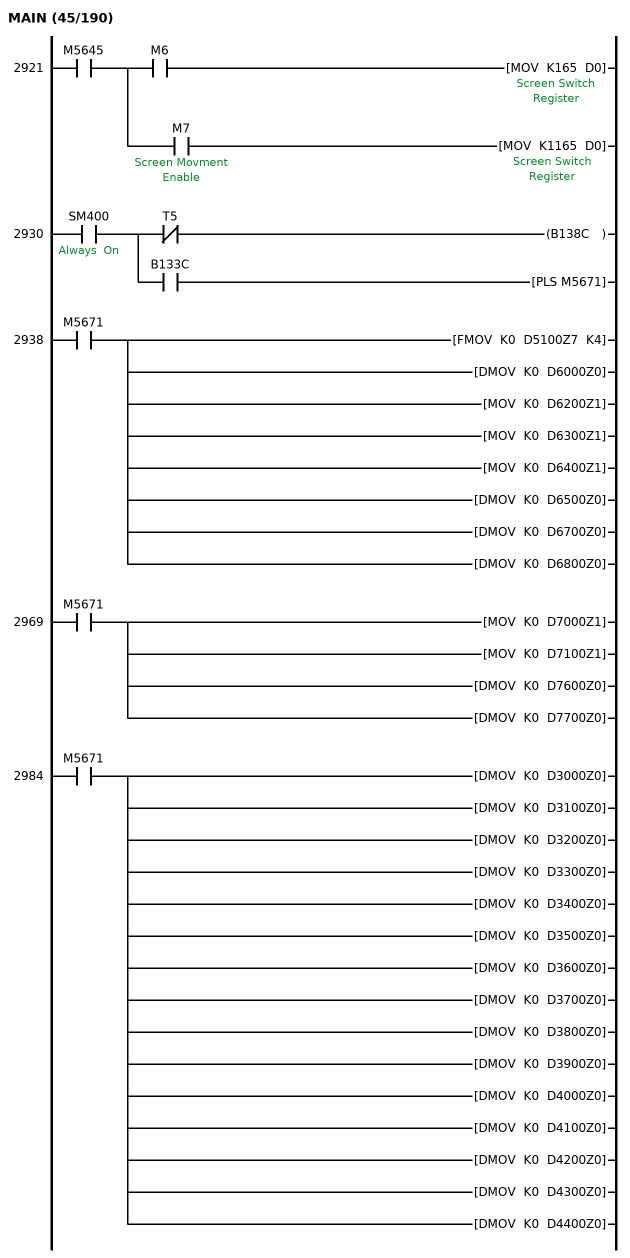
2921  LD      M5645
      MPS
      AND     M6
      MOV     K165 D0
      MPP
      AND     M7  ; Screen Movment Enable
      MOV     K1165 D0
2930  LD      SM400  ; Always  On
      MPS
      ANI     T5
      OUT     B138C
      MPP
      AND     B133C
      PLS     M5671
2938  LD      M5671
      FMOV    K0 D5100Z7 K4
      DMOV    K0 D6000Z0
      MOV     K0 D6200Z1
      MOV     K0 D6300Z1
      MOV     K0 D6400Z1
      DMOV    K0 D6500Z0
      DMOV    K0 D6700Z0
      DMOV    K0 D6800Z0
2969  LD      M5671
      MOV     K0 D7000Z1
      MOV     K0 D7100Z1
      DMOV    K0 D7600Z0
      DMOV    K0 D7700Z0
2984  LD      M5671
      DMOV    K0 D3000Z0
      DMOV    K0 D3100Z0
      DMOV    K0 D3200Z0
      DMOV    K0 D3300Z0
      DMOV    K0 D3400Z0
      DMOV    K0 D3500Z0
      DMOV    K0 D3600Z0
      DMOV    K0 D3700Z0
      DMOV    K0 D3800Z0
      DMOV    K0 D3900Z0
      DMOV    K0 D4000Z0
      DMOV    K0 D4100Z0
      DMOV    K0 D4200Z0
      DMOV    K0 D4300Z0
      DMOV    K0 D4400Z0
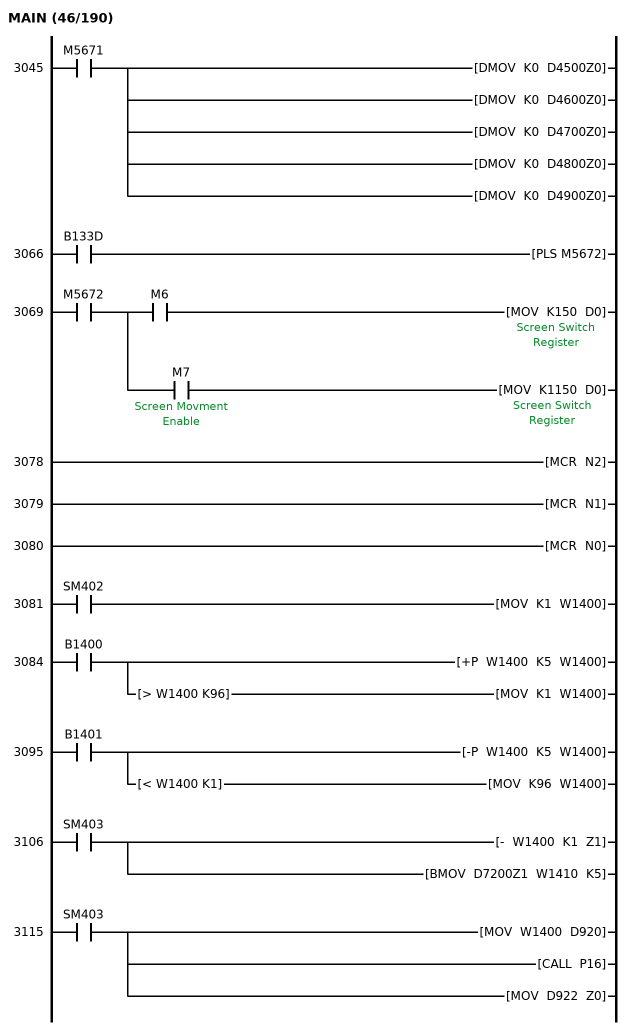
3045  LD      M5671
      DMOV    K0 D4500Z0
      DMOV    K0 D4600Z0
      DMOV    K0 D4700Z0
      DMOV    K0 D4800Z0
      DMOV    K0 D4900Z0
3066  LD      B133D
      PLS     M5672
3069  LD      M5672
      MPS
      AND     M6
      MOV     K150 D0
      MPP
      AND     M7  ; Screen Movment Enable
      MOV     K1150 D0
3078  MCR     N2
3079  MCR     N1
3080  MCR     N0
3081  LD      SM402
      MOV     K1 W1400
3084  LD      B1400
      +P      W1400 K5 W1400
      AND>    W1400 K96
      MOV     K1 W1400
3095  LD      B1401
      -P      W1400 K5 W1400
      AND<    W1400 K1
      MOV     K96 W1400
3106  LD      SM403
      -       W1400 K1 Z1
      BMOV    D7200Z1 W1410 K5
3115  LD      SM403
      MOV     W1400 D920
      CALL    P16
      MOV     D922 Z0
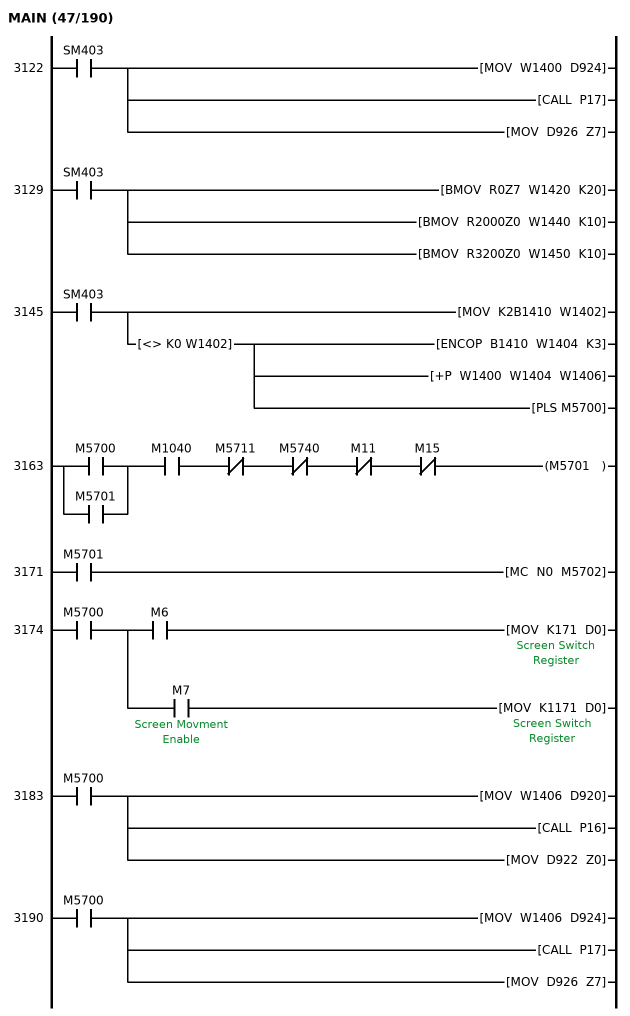
3122  LD      SM403
      MOV     W1400 D924
      CALL    P17
      MOV     D926 Z7
3129  LD      SM403
      BMOV    R0Z7 W1420 K20
      BMOV    R2000Z0 W1440 K10
      BMOV    R3200Z0 W1450 K10
3145  LD      SM403
      MOV     K2B1410 W1402
      AND<>   K0 W1402
      ENCOP   B1410 W1404 K3
      +P      W1400 W1404 W1406
      PLS     M5700
3163  LD      M5700
      OR      M5701
      AND     M1040
      ANI     M5711
      ANI     M5740
      ANI     M11
      ANI     M15
      OUT     M5701
3171  LD      M5701
      MC      N0 M5702
3174  LD      M5700
      MPS
      AND     M6
      MOV     K171 D0
      MPP
      AND     M7  ; Screen Movment Enable
      MOV     K1171 D0
3183  LD      M5700
      MOV     W1406 D920
      CALL    P16
      MOV     D922 Z0
3190  LD      M5700
      MOV     W1406 D924
      CALL    P17
      MOV     D926 Z7
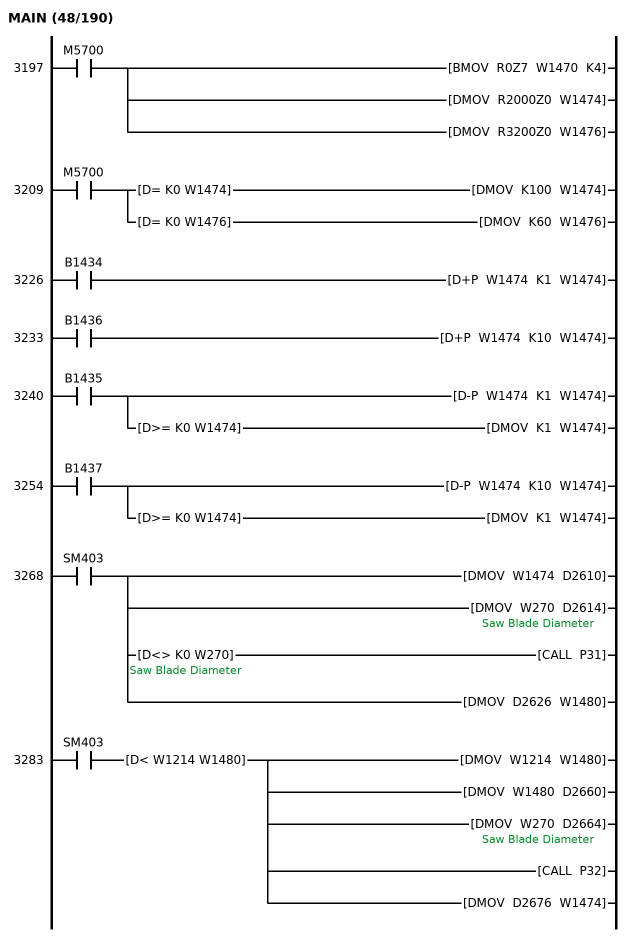
3197  LD      M5700
      BMOV    R0Z7 W1470 K4
      DMOV    R2000Z0 W1474
      DMOV    R3200Z0 W1476
3209  LD      M5700
      MPS
      ANDD=   K0 W1474
      DMOV    K100 W1474
      MPP
      ANDD=   K0 W1476
      DMOV    K60 W1476
3226  LD      B1434
      D+P     W1474 K1 W1474
3233  LD      B1436
      D+P     W1474 K10 W1474
3240  LD      B1435
      D-P     W1474 K1 W1474
      ANDD>=  K0 W1474
      DMOV    K1 W1474
3254  LD      B1437
      D-P     W1474 K10 W1474
      ANDD>=  K0 W1474
      DMOV    K1 W1474
3268  LD      SM403
      DMOV    W1474 D2610
      DMOV    W270 D2614
      MPS
      ANDD<>  K0 W270  ; Saw Blade Diameter
      CALL    P31
      MPP
      DMOV    D2626 W1480
3283  LD      SM403
      ANDD<   W1214 W1480
      DMOV    W1214 W1480
      DMOV    W1480 D2660
      DMOV    W270 D2664
      CALL    P32
      DMOV    D2676 W1474
